// TIA Portal V15 export
// export: Created 2018-05-30T14:06:23.9929541Z, ExportSetting WithDefaults, WithReadOnly, DisplayName Totally Integrated Automation Portal, DisplayVersion V15, DisplayName TIA Portal Openness, DisplayVersion V15, DisplayName STEP 7 Professional, DisplayVersion V15, DisplayName WinCC Professional, DisplayVersion V15
FUNCTION_BLOCK "BST_PIDAIN_400"   // FB25, STL
{ S7_Optimized_Access := 'FALSE' }
VERSION : 0.1
// stored: AutoNumber false, CodeModifiedDate 2018-05-30T14:05:05.4814636Z, CompileDate 2018-05-30T14:05:05.4814635Z, CreationDate 2018-05-30T13:57:54.5148136Z, InterfaceModifiedDate 2018-05-30T14:05:02.6553018Z, IsConsistent true, IsKnowHowProtected false, ISMultiInstanceCapable true, IsWriteProtected false, LibraryConformanceStatus The object is library-conformant., ModifiedDate 2018-05-30T14:05:05.4814636Z, ParameterModified 2018-05-30T14:05:02.6553018Z, StructureModified 2018-05-30T14:05:02.6553018Z, UDAEnableTagReadback false
   VAR_INPUT
      L_REMOTE : Bool;
      HMI_SP_INT : Real;
      L_AUT : Bool;
      HMI_MAN : Real;
      PV : Real;
      Set_SP : Bool;
      Set_Output : Bool;
   END_VAR
   VAR_OUTPUT
      PV_OUT : Real;
      QERR : Bool;
      LMN : Real;
   END_VAR
BEGIN
END_FUNCTION_BLOCK
